FUNCTION_BLOCK TmsMoverSequence
VAR_INPUT
	ThisMover : IMover;
	XtsTrack : IXtsTrack;
	StateMachine : IPmlStateMachine;
END_VAR
VAR_OUTPUT
END_VAR
VAR
END_VAR

END_FUNCTION_BLOCK

(* stored: Version 1.1.0.1, ProductVersion 3.1.4024.11
   POU TmsMoverSequence: Id {d0a7936d-1617-4a79-aef0-0b298f1ee6e2}, SpecialFunc None *)
